PROGRAM MAIN
VAR
	Logger : TcMessage_Ext := (LoggerLevel := TcEventSeverity.Verbose);
	iLogger : ITcMessage_Ext := Logger;
	bSendHello : BOOL;
	bSendError : BOOL;
END_VAR

IF bSendHello THEN
	iLogger.Send(Tc_Events.TestEventClass.Hello,' Bob');
	bSendHello := FALSE;	
END_IF

IF bSendError THEN
	iLogger.Send(Tc_Events.TestEventClass.Error, 'Oh dear');
	bSendError := FALSE;
END_IF

END_PROGRAM

(* stored: Version 1.1.0.1, ProductVersion 3.1.4024.11
   POU MAIN: Id {4fa24a04-fdb2-4ede-9fa0-d93eef268cc6}, SpecialFunc None *)
